{attribute 'qualified_only'}
VAR_GLOBAL
	stEL6021In  AT %I*	: EL6inData22B;		//**To EL6021 Inputs**
	stEL6021Out AT %Q*	: EL6outData22B;	//**To EL6021 Outputs**
END_VAR

(* stored: Version 1.1.0.1, ProductVersion 3.1.4024.12
   GVL DistanceSensor: Id {baca80ce-a208-42b3-b2b4-8a03c96bd8b9} *)
